// TIA Portal V20 export
// export: Created 2025-12-01T14:57:09.4995079Z, ExportSetting None, DisplayName Totally Integrated Automation Portal, DisplayVersion V20 Update 3, DisplayName TIA Portal Openness, DisplayVersion V20 Update 3, DisplayName TIA Portal Version Control Interface, DisplayVersion V20 Update 3, DisplayName STEP 7 Professional, DisplayVersion V20 Update 3, DisplayName STEP 7 Safety, DisplayVersion V20 Update 2, DisplayName WinCC Basic/Comfort/Advanced, DisplayVersion V20 Update 3, DisplayName WinCC Professional, DisplayVersion V20 Update 3, DisplayName WinCC Unified, DisplayVersion V20 Update 3
FUNCTION "FC720_BuscarUT_EnMesa" : Void   // FC720, LAD
TITLE = "BuscarUT" - Buscar donde esta una UT determinada
{ S7_Optimized_Access := 'FALSE' }
AUTHOR : TRACKING
NAME : 20130301
VERSION : 3.0
// stored: AutoNumber false, SetENOAutomatically false
   VAR_INPUT
      Mckey : UDInt;   // Mckey de la UT
      MesaActual : UInt;   // Mesa Actual de la UT (En PLC)
   END_VAR
   VAR_OUTPUT
      NumeroUT : UInt;   // Donde esta la UT en DB_DatosUT
   END_VAR
   VAR_TEMP
      Mesa : UInt;   // Mesa
      NumUT : UInt;   // Numero UT
      ColaMckey : UInt;   // Numero de Cola de Mckey
   END_VAR
BEGIN

NETWORK
TITLE = Inicilizar
// - Iniciliza numero de DB's
// - Iniciliza variables internas
///////////////////////////////////////////////////////////////////////////////
// Inicializa las variables
      L     0;  // No existe Mckey
      T     #NumeroUT;
      T     #NumUT;

      L     #MesaActual;  // Ver que mesa es
      T     #Mesa;



NETWORK
TITLE = Bucle de la Busqueda por Mckey
// Recorre toda la cola de ordenacion de Mckey buscando la UT
// - De aqui no tiene que pasar
///////////////////////////////////////////////////////////////////////////////
///////////////////////////////////////////////////////////////////////////////
// Busqueda del Mckey en DB_OrdenadoMckey
      L     #Mckey;
      L     10000;  // 10.000 Colas de Mckey
      MOD;
      T     #ColaMckey;  // Numero de la Cola de Mckey


///////////////////////////////////////////////////////////////////////////////
      L     "DB811_ColasMckeys".Colas_Mckey[#ColaMckey].UT_PrimerMckey;
      T     #NumUT;

      L     #NumUT;
      L     0;
      ==I;
      JC    Busqueda_PorMesaActual;  // Hay UT's en la Cola de Mckey ?


///////////////////////////////////////////////////////////////////////////////
///////////////////////////////////////////////////////////////////////////////
///////////////////////////////////////////////////////////////////////////////
// Recorro las UT de la Cola de Mckey
InicoBucle_Mckey:NOP   0;
      L     "DB812_UTs_Control".UT[#NumUT].Mckey;
      L     #Mckey;  // Si es mismo MCkey
      ==D;
      JC    FinalFuncion;


///////////////////////////////////////////////////////////////////////////////
// ----- No es mismo Mckey
//       Mirar la siguiente de la Cola de Mckey
      L     "DB811_ColasMckeys".MckeyUT[#NumUT].UT_SiguienteMcKey;
      T     #NumUT;

      L     #NumUT;  // Hay mas UT's en la Cola de Mckey
      L     0;
      ==I;
      JC    Busqueda_PorMesaActual;  // No existe UT
      JU    InicoBucle_Mckey;



NETWORK
TITLE = Bucle de la Busqueda por Mesa
// Recorre toda la cola de la mesa buscando la UT
// - Si llega aqui malamente
///////////////////////////////////////////////////////////////////////////////
///////////////////////////////////////////////////////////////////////////////
///////////////////////////////////////////////////////////////////////////////
// Mirar antes de buscar si pasa Mesa
Busqueda_PorMesaActual:NOP   0;
      L     #Mesa;
      L     0;
      ==I;
      JC    Busqueda_PorListaUTs;


///////////////////////////////////////////////////////////////////////////////
///////////////////////////////////////////////////////////////////////////////
///////////////////////////////////////////////////////////////////////////////
// Empiezo a recorrer los datos de UT en la Mesa
// Miro primero si hay alguna UT en la Mesa
      L     "DB810_ColasMesas".Colas[#Mesa].UT_PrimeraMesa;
      T     #NumUT;

      L     #NumUT;
      L     0;
      ==I;
      JC    Busqueda_PorListaUTs;  // Hay UT's en la Mesa


///////////////////////////////////////////////////////////////////////////////
// Recorro las UT de las mesas
InicioBucle_MesaActual:NOP   0;
      L     "DB812_UTs_Control".UT[#NumUT].Mckey;
      L     #Mckey;  // Si es mismo MCkey
      ==D;
      JC    FinalFuncion;


///////////////////////////////////////////////////////////////////////////////
// ----- No es mismo Mckey
//       Mirar la siguinte de la Mesa
      L     "DB812_UTs_Control".UT[#NumUT].UT_SiguienteMesa;
      T     #NumUT;

      L     #NumUT;  // Hay mas UT's en la Mesa
      L     0;
      ==I;
      JC    Busqueda_PorListaUTs;  // No existe UT
      JU    InicioBucle_MesaActual;



NETWORK
TITLE = Bucle de la Busqueda por UT's directamente
// Recorre todas las UT's buscando la UT
// Si llega aqui mala cosa - muy muy malamente
///////////////////////////////////////////////////////////////////////////////
///////////////////////////////////////////////////////////////////////////////
///////////////////////////////////////////////////////////////////////////////
Busqueda_PorListaUTs:NOP   0;
      L     1;
      T     #NumUT;  // Inicializar


///////////////////////////////////////////////////////////////////////////////
// Recorro la  Lista de UTs
InicioBucle_ListaUTs:NOP   0;
      L     "DB812_UTs_Control".UT[#NumUT].Mckey;
      L     #Mckey;  // Si es mismo MCkey
      ==D;
      JC    FinalFuncion;


///////////////////////////////////////////////////////////////////////////////
// ----- No es mismo Mckey
//       Mirar la siguinte UT
      L     #NumUT;  // A la siguiente UT
      L     1;
      +I;
      T     #NumUT;

      L     #NumUT;
      L     "CTE_MaxUTs";
      >I;
      JC    FinalBucle_ListaUTs;
      JU    InicioBucle_ListaUTs;


///////////////////////////////////////////////////////////////////////////////
///////////////////////////////////////////////////////////////////////////////
///////////////////////////////////////////////////////////////////////////////
FinalBucle_ListaUTs:NOP   0;
      L     0;  // No se ha encontrado
      T     #NumUT;
      JU    FinalFuncion;



NETWORK
TITLE = Finalizar funcion
// Devuelve el Numero de UT
///////////////////////////////////////////////////////////////////////////////
///////////////////////////////////////////////////////////////////////////////
///////////////////////////////////////////////////////////////////////////////
FinalFuncion:NOP   0;
      L     #NumUT;
      T     #NumeroUT;  // Devolucion de la funcion


END_FUNCTION
